//---------------------------------------------------------------------------------------------------------------
//
//  HAUD 2023.03.27
//
//  TR08
//  - XTS_TRANSPORT_LAYER
//
//  fb_Process
//  - grouping of xts stations to sync start process
//  - nFirst to nLast xts stations are checked for starting process simultaneously
//  - basic preparation of station target index in PrepareTarget()
//  - handshake with station control for mover transport through station
//
//---------------------------------------------------------------------------------------------------------------
// This SOFTWARE is provided as an Exemple by THE PROVIDER "as is" and "with all faults." THE PROVIDER makes no 
// representations or warranties of any kind concerning the safety, suitability, lack of viruses, inaccuracies, 
// typographical errors, or other harmful components of this SOFTWARE. There are inherent dangers in the use of 
// any software, and you are solely responsible for determining whether this SOFTWARE is compatible with your 
// equipment and other software installed on your equipment. You are also solely responsible for the protection 
// of your equipment and backup of your data, and THE PROVIDER will not be liable for any damages you may suffer 
// in connection with using, modifying, or distributing this SOFTWARE.
//---------------------------------------------------------------------------------------------------------------
FUNCTION_BLOCK fb_Process IMPLEMENTS I_ExternControl_Process
VAR
  _eType                      : E_PROCESS_TYPE;   // types of process: SINGLE, PARALLEL, SERIAL, DISTRIBUTOR
  _sCheck                     : STRING;

  _eProcessCmd                : E_STATION_CTRL;   // control from property
  _eProcessState              : E_STATION_STATE;  // state   to   property

  {attribute 'displaymode':='bin'}
  _wEnableProcess             : DWORD; // control sets bits to switch on stations
  _bEnabledStation            : POINTER TO ARRAY[1..XTS_Parameter.MAX_STATION]  OF BOOL; // information about all enabled xts stations

  // xts stations
  _stCtrl                     : POINTER TO ARRAY[1..XTS_Parameter.MAX_STATION]  OF ST_STATION_CTRL;
  _stState                    : POINTER TO ARRAY[1..XTS_Parameter.MAX_STATION]  OF ST_STATION_STATE;

  // who is included in process
  // _nFirst to _nLast MUST be in closed consecutive order
  _nStation,
  _nStationCount,
  _nFirstStation,
  _nLastStation               : UINT;

  // work vars for writing onto _stCtrl[nStation].nTargetStation
  _nTarget,
  _nFirstTarget,
  _nLastTarget                : UINT;   // for parallel process xts stations and the last xts station in serial process

  _nSerialTarget              : ARRAY[1..XTS_Parameter.MAX_STATION]  OF UINT; // serial targets within process

  _nPreparedTarget            : ARRAY[1..XTS_Parameter.MAX_MOVER]  OF UINT;   // targets for parallel and single process

  // bitmasks for station states in CycleStation()
  {attribute 'displaymode':='bin'}
  _wEnable                    : DWORD;   // commanded enable of xts station
  {attribute 'displaymode':='bin'}
  _wEnter                     : DWORD;   // mover asking for entry into xts station
  {attribute 'displaymode':='bin'}
  _wStart                     : DWORD;   // xts station asking for process handshake
  {attribute 'displaymode':='bin'}
  _wLeave                     : DWORD;   // xts station wants to send out mover
  {attribute 'displaymode':='bin'}
  _wQueue                     : DWORD;   // mover was entered into xts station list
  {attribute 'displaymode':='bin'}
  _wMoverInStation            : DWORD;   // mover entry was granted, mover is now in station
  {attribute 'displaymode':='bin'}
  _wError                     : DWORD;   // minor error, must be fixed by _stCtrl[nStation]
  {attribute 'displaymode':='bin'}
  _wErrorFatal                : DWORD;   // fatal error, must be fixed by debugging
  {attribute 'displaymode':='bin'}
  _wTargetId                  : DWORD;   // nTargetStation > 0 in _stDtrl[nStation].nTargetStation

  {attribute 'displaymode':='bin'}
  _TargetMask                 : DWORD;   // bit positions correspond to index of xts station
 
  _bNext                      : BOOL;

  _nProcessPerMinute          : uint; // sum of all xts stations output per minute in process
  _rtrigProcess               : ARRAY[1..XTS_Parameter.MAX_STATION] OF Tc2_Standard.R_TRIG;
  _tonPartsPerMinute          : Tc2_Standard.TON;

  _nMoverPerMinute            : POINTER TO ARRAY[1..XTS_Parameter.MAX_STATION]  OF UINT;
  _nMoverCount,
  _nMoverCountOld             : ARRAY[1..XTS_Parameter.MAX_STATION]  OF UINT;

  _eDistributorTarget         : E_PROGRESS;

END_VAR

METHOD private Check : BOOL

IF (_nFirstStation < 1) OR
   (_nFirstStation > MAX_STATION)
THEN
  _sCheck                     := '_nFirstStation out of bounds';
  RETURN;
END_IF

IF (_nLastStation < 1) OR
   (_nLastStation > MAX_STATION)
THEN
  _sCheck                     := '_nLastStation out of bounds';
  RETURN;
END_IF

IF (_nFirstTarget < 1) OR
   (_nFirstTarget > MAX_STATION)
THEN
  _sCheck                     := '_nFirstTarget out of bounds';
  RETURN;
END_IF

IF (_nLastTarget < 1) OR
   (_nLastTarget > MAX_STATION)
THEN
  _sCheck                     := '_nLastTarget out of bounds';
  RETURN;
END_IF

IF NOT (_stCtrl  <> 0)
THEN
  _sCheck                     := '_stCtrl: missing pointer';
  RETURN;
END_IF

IF NOT (_stState <> 0)
THEN
  _sCheck                     := '_stState: missing pointer';
  RETURN;
END_IF

IF NOT (_bEnabledStation  <> 0)
THEN
  _sCheck                     := '_bEnableStation: missing pointer';
  RETURN;
END_IF

IF not (_nMoverPerMinute <> 0)
THEN
  _sCheck                     := '_nMoverPerMinute: missing pointer';
  RETURN;
END_IF

_nStationCount                := _nLastStation - _nFirstStation + 1;

IF (_nStationCount < 1) OR
   (_nStationCount > (SIZEOF(WORD)*8))
THEN
  _sCheck                     := '_nStationCount out of bounds';
  RETURN;
END_IF


_sCheck                       := TO_STRING(E_PROGRESS.PROGRESS_DONE);
Check                         := TRUE;
END_METHOD

METHOD Cycle
VAR_INST
  _nStn     : uint;
END_VAR
IF NOT Check() THEN RETURN; END_IF


//-----------------------------------------------------------------------------
// collect state information from xts stations
// state information is collected in Masks (WORD), 
// every bit represents one XTS station in process
//-----------------------------------------------------------------------------
//  _wEnable                        : enable cmd was given to xts station
//  _wEnter                         : a mover is requesting entry
//  _wStart                         : mover has arrived and xts station is ready
//  _wLeave                         : xts station wants to send mover out
//  _wQueue                         : somebody's waiting
//  _wMoverInStation                : mover is in station
//  _wError                         : error state for handshake
//  _wErrorFatal                    : error state for severe problems (debugging required)
//  _wTargetId                      : Ctrl.nTargetStation > 0
//  _wMoverInQueueSerial            : SERIAL process: bits to check whether a mover is waiting to be processed
//
CycleStation();                     // get state information from all XtsStations in process
//-----------------------------------------------------------------------------
//-----------------------------------------------------------------------------
//  E_STATION_CTRL.STATION_INIT: hard reset of process and XtsStations
//-----------------------------------------------------------------------------
CASE _eProcessCmd                   // check input property
OF
  E_STATION_CTRL.STATION_INIT:      // commanded init from ctrl
    CASE _eType
    OF
      E_PROCESS_TYPE.SERIAL:
        InitSerialTargets();
    END_CASE
    Init();                         RETURN; // rest you will, return you must
END_CASE
//-----------------------------------------------------------------------------
// E_STATION_STATE.STATION_INIT: pass through here and switch off XtsStations
//-----------------------------------------------------------------------------
CASE _eProcessState                 // check output property
OF
  E_STATION_STATE.STATION_INIT:     // xts station empty, disabled by default
    _eProcessState                  := E_STATION_STATE.STATION_DISABLE;
    FOR _nStn := _nLastStation TO _nFirstStation BY(-1) 
    DO
      _stCtrl^[_nStn].eCmd          := E_STATION_CTRL.STATION_DISABLE;
    END_FOR

END_CASE
//-----------------------------------------------------------------------------
//  E_STATION_STATE.STATION_DISABLE: wait for enable from flow control
//-----------------------------------------------------------------------------
CASE _eProcessState                 // check output property
OF
  E_STATION_STATE.STATION_DISABLE:  // check for enable command
    IF (_eProcessCmd = E_STATION_CTRL.STATION_ENABLE)
    THEN
      _eProcessState                := E_STATION_STATE.STATION_ENABLE;

      FOR _nStn := _nLastStation TO _nFirstStation BY(-1) 
      DO
          _stCtrl^[_nStn].eCmd      := E_STATION_CTRL.STATION_ENABLE;
      END_FOR
    END_IF
END_CASE
//-----------------------------------------------------------------------------
//  E_STATION_STATE.STATION_ENABLE: check Cmd and wait for XtsStations to be enabled
//-----------------------------------------------------------------------------
CASE _eProcessState
OF
  E_STATION_STATE.STATION_ENABLE:
    CASE _eProcessCmd
    OF
      E_STATION_CTRL.STATION_DISABLE:
        _eProcessState              := E_STATION_STATE.STATION_INIT;

      E_STATION_CTRL.STATION_ENABLE:
        IF (_wEnable = _wEnableProcess)
        THEN
          InitSerialTargets();
          _eProcessState            := E_STATION_STATE.STATION_DETECT_MOVER;
        END_IF
    END_CASE
END_CASE
//-----------------------------------------------------------------------------
// E_STATION_STATE.STATION_DETECT_MOVER: wait for any XtsStation to 
//                                       have a mover ready to enter
//-----------------------------------------------------------------------------
CASE _eProcessState
OF
  E_STATION_STATE.STATION_DETECT_MOVER:
    CASE _eProcessCmd
    OF
      E_STATION_CTRL.STATION_DISABLE:
        _eProcessState              := E_STATION_STATE.STATION_INIT;

      E_STATION_CTRL.STATION_ENABLE:
        IF (_wEnter > 0)            // at least one mover is asking for entry
        THEN
          _eDistributorTarget       := E_PROGRESS.PROGRESS_INVALID;

                                    // switch process state in order to tell process control
          _eProcessState            := E_STATION_STATE.STATION_MOVER_ENTER;
        END_IF
    END_CASE
END_CASE
//-----------------------------------------------------------------------------
//  E_STATION_STATE.STATION_MOVER_ENTER: check if infeed conditions are met, 
//                                       depending on type of process
//                                       Cmd from input (flow control)
//-----------------------------------------------------------------------------
CASE _eProcessState
OF
  E_STATION_STATE.STATION_MOVER_ENTER:
    CASE _eProcessCmd               // check input property
    OF
      E_STATION_CTRL.STATION_DISABLE:
        _eProcessState              := E_STATION_STATE.STATION_INIT;

      E_STATION_CTRL.STATION_MOVER_ENTER:
        FOR _nStn := _nLastStation TO _nFirstStation BY(-1) 
        DO
          CASE _stState^[_nStn].eState
          OF
          E_STATION_STATE.STATION_MOVER_ENTER,
          E_STATION_STATE.STATION_MOVER_IN_TARGET,
          E_STATION_STATE.STATION_PROCESS_START:
            IF GetBitDWord(_wEnter, (_nStn - _nFirstStation))
            THEN
              _stCtrl^[_nStn].eCmd  := E_STATION_CTRL.STATION_MOVER_ENTER;
            END_IF
          END_CASE
        END_FOR

        CASE _eType
        OF
          E_PROCESS_TYPE.PARALLEL_STRICT:
            IF (_wStart = _wEnable) // all who are enabled must have mover, in order to continue
            THEN
              _eProcessState        := E_STATION_STATE.STATION_PROCESS_START;
            END_IF

          E_PROCESS_TYPE.PARALLEL: 
            IF (_wStart = _wEnter)
            THEN
              _eProcessState        := E_STATION_STATE.STATION_PROCESS_START;
            END_IF

          E_PROCESS_TYPE.SERIAL:    // all who have work to do must have mover, in order to continue
            IF (_wMoverInStation > 0)
            THEN
              IF (_wStart = _wMoverInStation)
              THEN
                _eProcessState      := E_STATION_STATE.STATION_PROCESS_START;
              END_IF
            END_IF
        ELSE
          _eProcessState            := E_STATION_STATE.STATION_PROCESS_START;
        END_CASE

      E_STATION_CTRL.STATION_MOVER_SEND:  // flow control decided to skip process
        FOR _nStn := _nLastStation TO _nFirstStation BY(-1) 
        DO
          IF _bEnabledStation^[_nStn] AND 
             GetBitDWord(_wQueue, (_nStn-_nFirstStation))
          THEN
            IF (_TargetMask > 0)
            THEN
              // station is enabled AND has a mover in Queue to send
              _stCtrl^[_nStn].eCmd    := E_STATION_CTRL.STATION_MOVER_SEND;
            END_IF
          END_IF
        END_FOR
        IF (_wLeave > 0)            // wait for XtsStation to switch to outfeed
        THEN
          IF (_TargetMask > 0)
          THEN
            _eDistributorTarget       := DistributorTarget(_TargetMask);         // prepare target for mover
            IF (_eDistributorTarget = E_PROGRESS.PROGRESS_DONE)
            THEN
              _wStart                 := _wLeave;
              _eProcessState          := E_STATION_STATE.STATION_CHECK;
            END_IF
          END_IF
        END_IF 
    END_CASE
END_CASE
//-----------------------------------------------------------------------------
// synced process handshake on all stations in process
//-----------------------------------------------------------------------------
CASE _eProcessState                 // check output property
OF
  E_STATION_STATE.STATION_PROCESS_START:
    CASE _eType                     // decision for synced start varies for e_process_type
    OF
      E_PROCESS_TYPE.SERIAL:        // serial process must have had a mover waiting, which is now processed
      CASE _eProcessCmd             // check command input property
      OF
        E_STATION_CTRL.STATION_PROCESS_START,
        E_STATION_CTRL.STATION_PROCESS_DONE:
            IF (_wStart = _wMoverInStation)
            THEN
              _eProcessState          := E_STATION_STATE.STATION_PROCESS_DONE;
              FOR _nStn := _nLastStation TO _nFirstStation BY(-1) 
              DO
                // check for correct state on XtsStation
                CASE _stState^[_nStn].eState
                OF
                E_STATION_STATE.STATION_PROCESS_START:
                  _stCtrl^[_nStn].eCmd  := _eProcessCmd;
                END_CASE
              END_FOR
            END_IF
      END_CASE
    ELSE
      CASE _eProcessCmd             // check command input property
      OF
        E_STATION_CTRL.STATION_PROCESS_START,
        E_STATION_CTRL.STATION_PROCESS_DONE:
          IF (_wStart = _wEnter)
          THEN
            _eProcessState          := E_STATION_STATE.STATION_PROCESS_DONE;
            FOR _nStn := _nLastStation TO _nFirstStation BY(-1) 
            DO
              // check for correct state on XtsStation
              CASE _stState^[_nStn].eState
              OF
              E_STATION_STATE.STATION_PROCESS_START:
                _stCtrl^[_nStn].eCmd  := _eProcessCmd;
              END_CASE
            END_FOR
          END_IF
      END_CASE
    END_CASE
END_CASE
//-----------------------------------------------------------------------------
// synced process handshake on all stations in process
//-----------------------------------------------------------------------------
CASE _eProcessState                 // check output property
OF
  E_STATION_STATE.STATION_PROCESS_DONE:
    CASE _eProcessCmd               // check command input property
    OF
      E_STATION_CTRL.STATION_PROCESS_DONE: 
        FOR _nStn := _nLastStation TO _nFirstStation BY(-1) 
        DO
          _stCtrl^[_nStn].eCmd      := E_STATION_CTRL.STATION_PROCESS_DONE;
        END_FOR
        IF (_wLeave > 0)            // _wLeave tells us that xts station has mover to send
        THEN
          CASE _eType
          OF
            E_PROCESS_TYPE.SERIAL:
              _eProcessState        := E_STATION_STATE.STATION_CHECK;
              IF (_stState^[_nLastStation].nMoverId > 0)
              THEN
                PrepareLastSerialTarget();     // target for last xts station in serial process
              END_IF
    
              FOR _nStn := (_nLastStation - 1) TO _nFirstStation BY(-1) 
              DO
                _stCtrl^[_nStn].nTargetStation    := TO_USINT(_nSerialTarget[_nStn]);
              END_FOR
          ELSE
              IF (_TargetMask > 0)
              THEN
                ParallelTargets(_TargetMask);
                _eProcessState      := E_STATION_STATE.STATION_CHECK;
              END_IF
          END_CASE
        END_IF
    END_CASE
END_CASE
//-----------------------------------------------------------------------------
//-----------------------------------------------------------------------------
CASE _eProcessState
OF
  E_STATION_STATE.STATION_CHECK:    // TODO: implement procedure for target plausibility
    IF (_wTargetId > 0)             // simple check any target before switching to outfeed
    THEN
       _eProcessState               := E_STATION_STATE.STATION_MOVER_OUT;
(*
    ELSE                            // in case of invalid target, wait here for retry
      CASE _eType                   // retry varies for e_process_type
      OF
        E_PROCESS_TYPE.DISTRIBUTOR:
          IF (_eProcessCmd = E_STATION_CTRL.STATION_ENABLE)
          THEN
            // only distributor can land here directly; retry mover infeed
            _eProcessState          := E_STATION_STATE.STATION_MOVER_ENTER;
          END_IF
      ELSE
          IF (_eProcessCmd = E_STATION_CTRL.STATION_PROCESS_START)
          THEN
            // all other e_process_type must go back to process handshake
            _eProcessState          := E_STATION_STATE.STATION_PROCESS_DONE;
          END_IF
      END_CASE
*)
    END_IF
END_CASE
//-----------------------------------------------------------------------------
//-----------------------------------------------------------------------------
CASE _eProcessState
OF
  E_STATION_STATE.STATION_MOVER_OUT:
    IF (_wLeave = 0)                // all movers are gone
    THEN
      _eProcessState                := E_STATION_STATE.STATION_MOVER_GONE;

    ELSIF (_wLeave = _wStart)       // wait for everybody to be ready for send out
    THEN
      IF (_eProcessCmd = E_STATION_CTRL.STATION_MOVER_OUT)
      THEN
        FOR _nStn := _nLastStation TO _nFirstStation BY(-1) 
        DO
          CASE _stState^[_nStn].eState  // double check valid xts station state
          OF
            E_STATION_STATE.STATION_MOVER_OUT:
              IF (_stCtrl^[_nStn].nTargetStation > 0) // double check ticket on ctrl struct
              THEN
                _stCtrl^[_nStn].eCmd  := E_STATION_CTRL.STATION_MOVER_OUT;
              END_IF
          END_CASE
        END_FOR
      END_IF
    END_IF
END_CASE
//-----------------------------------------------------------------------------
//-----------------------------------------------------------------------------
CASE _eProcessState
OF
  E_STATION_STATE.STATION_MOVER_GONE:   // station is empty, quit mover gone and go back to the beginning
    FOR _nStn := _nLastStation TO _nFirstStation BY(-1) 
    DO
      _stCtrl^[_nStn].nTargetStation := 0;
      _stCtrl^[_nStn].eCmd      := E_STATION_CTRL.STATION_MOVER_GONE;
    END_FOR
    _eProcessState              := E_STATION_STATE.STATION_INIT;
END_CASE
END_METHOD

METHOD PRIVATE CycleStation
VAR
  _k                  : UINT;
END_VAR
IF NOT Check() THEN RETURN; END_IF

_wError                                   :=
_wErrorFatal                              := 0;

FOR _nStation := _nLastStation TO _nFirstStation BY(-1) 
DO
  // copy bit for enable station from input word to global array in GVL_PROCESS,
  //  - other processes read enabled state on mover out (PrepareTarget)
  _bEnabledStation^[_nStation]            := GetBitDWord(_wEnableProcess, (_nStation-_nFirstStation));

  IF (_stCtrl^[_nStation].nTargetStation > 0)
  THEN
    _wTargetId                            := SetBitDWord(_wTargetId,  (_nStation-_nFirstStation));
  ELSE
    _wTargetId                            := DelBitDWord(_wTargetId,  (_nStation-_nFirstStation));
  END_IF

  IF (_stState^[_nStation].nMoverId > 0)
  THEN
    _wMoverInStation                      := SetBitDWord(_wMoverInStation,  (_nStation-_nFirstStation));
  ELSE
    _wMoverInStation                      := DelBitDWord(_wMoverInStation,  (_nStation-_nFirstStation));
  END_IF

  IF (_stState^[_nStation].nQueue > 0)
  THEN
    _wQueue                               := SetBitDWord(_wQueue,  (_nStation-_nFirstStation));
  ELSE
    _wQueue                               := DelBitDWord(_wQueue,  (_nStation-_nFirstStation));
  END_IF

  CASE _stCtrl^[_nStation].eCmd
  OF
    E_STATION_CTRL.STATION_INIT:
      _stCtrl^[_nStation].nTargetStation  := 0;
      _wEnable                            := DelBitDWord(_wEnable, (_nStation-_nFirstStation));
      _wEnter                             := DelBitDWord(_wEnter,  (_nStation-_nFirstStation));
      _wStart                             := DelBitDWord(_wStart,  (_nStation-_nFirstStation));
      _wLeave                             := DelBitDWord(_wLeave,  (_nStation-_nFirstStation));

    E_STATION_CTRL.STATION_ENABLE:
      _wEnable                            := SetBitDWord(_wEnable, (_nStation-_nFirstStation));
  END_CASE

  CASE _stState^[_nStation].eState
  OF
    E_STATION_STATE.STATION_DISABLE:
      _wEnter                             := DelBitDWord(_wEnter,  (_nStation-_nFirstStation));

    E_STATION_STATE.STATION_MOVER_ENTER,
    E_STATION_STATE.STATION_MOVER_IN_TARGET:
      _wEnter                             := SetBitDWord(_wEnter,  (_nStation-_nFirstStation));
  
    E_STATION_STATE.STATION_PROCESS_START,
    E_STATION_STATE.STATION_PROCESS_DONE:
      _wStart                             := SetBitDWord(_wStart,  (_nStation-_nFirstStation));
  
    E_STATION_STATE.STATION_MOVER_OUT:
      _wLeave                             := SetBitDWord(_wLeave,  (_nStation-_nFirstStation));


    E_STATION_STATE.STATION_MOVER_GONE:
      _stCtrl^[_nStation].nTargetStation  := 0;
      _wStart                             := DelBitDWord(_wStart,  (_nStation-_nFirstStation));
      _wLeave                             := DelBitDWord(_wLeave,  (_nStation-_nFirstStation));
      _wEnable                            := DelBitDWord(_wEnable, (_nStation-_nFirstStation));
      _wEnter                             := DelBitDWord(_wEnter,  (_nStation-_nFirstStation));


    E_STATION_STATE.STATION_ERROR_LIST_STATION_ID_WRONG,  // wrong station ID in mover ticket (nTargetId written by preceeding station/process)
    E_STATION_STATE.STATION_ERROR_OUTFEED_TARGET_INVALID, // write correct target on station Ctrl.nTargetStation
    E_STATION_STATE.STATION_ERROR_INFEED_ERROR,           // clear mover error via Ctrl/State interface and retry on XTS station directly
    E_STATION_STATE.STATION_ERROR_OUTFEED_ERROR:          // clear mover error via Ctrl/State interface and retry on XTS station directly
      _wError                             := SetBitDWord(_wError,      (_nStation-_nFirstStation));

    E_STATION_STATE.STATION_ERROR_FATAL:
      _wErrorFatal                        := SetBitDWord(_wErrorFatal, (_nStation-_nFirstStation));

  END_CASE
END_FOR


_nProcessPerMinute          := 0;
// get mover counter
FOR _k := _nLastStation TO _nFirstStation BY(-1) 
DO
  _rtrigProcess[_k](
                  CLK       := (_stCtrl^[_k].eCmd = E_STATION_CTRL.STATION_MOVER_OUT));

  IF _rtrigProcess[_k].Q
  THEN
    _nMoverCount[_k]        := _nMoverCount[_k] + 1;
  END_IF
  
  IF _tonPartsperMinute.Q
  THEN
    _nMoverPerMinute^[_k]   := _nMoverCount[_k] - _nMoverCountOld[_k];
    _nMoverCountOld  [_k]   := _nMoverCount[_k];
  END_IF
  _nProcessPerMinute        := _nProcessPerMinute + _nMoverPerMinute^[_k]; 
END_FOR

IF _tonPartsperMinute.q
THEN
  _tonPartsperMinute(
                  IN        :=FALSE);
END_IF

_tonPartsperMinute(
                  IN        := TRUE, 
                  PT        := T#60S);
END_METHOD

METHOD PUBLIC DelBitDWord : DWORD
VAR_INPUT
  inVal   : DWORD;
  bitNo   : DWORD;
END_VAR
VAR
  wConst : DWORD := 1;
END_VAR
IF ( inVal AND SHL( wConst,bitNo MOD 16 ) ) > 0 THEN
  DelBitDWord := inVal XOR (SHL( wConst,bitNo MOD 16 ));
ELSE
  DelBitDWord := inVal;
END_IF
END_METHOD

METHOD DistributorTarget : e_progress
VAR_INPUT
  wTarget         : DWORD; // bits for target stations to be used
END_VAR
VAR_INST
  _eResult        : E_PROGRESS;
  {attribute 'displaymode':='bin'}
  _wtg            : DWORD;
END_VAR
IF NOT Check() THEN RETURN; END_IF
_wtg := wTarget;

// check if target station is enabled
IF GetBitDWord(wTarget, (_nTarget))
THEN
  _nPreparedTarget[_stState^[_nFirstStation].nMoverId]  := _nLastTarget - _nTarget;
  _stCtrl^[_nFirstStation].nTargetStation               := TO_USINT(_nLastTarget - _nTarget);
  _eResult                                              := E_PROGRESS.PROGRESS_DONE;
ELSE
  _eResult                                              := e_progress.PROGRESS_BUSY;
END_IF

_nTarget                      := _nTarget + 1;
IF (_nLastTarget - _nTarget < _nFirstTarget)
THEN
  _nTarget                    := 0;
END_IF

DistributorTarget                                       := _eResult;
END_METHOD

PROPERTY EnabledStation : POINTER TO ARRAY[1..XTS_Parameter.MAX_STATION]  OF bool;
SET
_bEnabledStation := EnabledStation;
END_SET
END_PROPERTY

PROPERTY EnableProcess : dword
GET
EnableProcess := _wEnableProcess;
END_GET
SET
_wEnableProcess := EnableProcess;
END_SET
END_PROPERTY

METHOD PUBLIC GetBitDWord : BOOL
VAR_INPUT
  inVal   : DWORD;
  bitNo   : DINT;
END_VAR
VAR
  wConst : DWORD := 1;
END_VAR
IF ( inVal AND SHL( wConst,DINT_TO_SINT(bitNo) MOD 32 ) ) > 0
THEN
  GetBitDWord := TRUE;
ELSE
  GetBitDWord := FALSE;
END_IF
END_METHOD

METHOD PUBLIC Init : BOOL
VAR
  _nStn     : UINT;
END_VAR
IF NOT (_nLastStation   > 0) OR
   NOT (_nFirstStation  > 0) OR
   NOT (_nLastStation   < MAX_STATION+1) OR
   NOT (_nFirstStation  < MAX_STATION+1)
THEN
  Init := FALSE;
  _eProcessState                := E_STATION_STATE.STATION_NO_INIT;
ELSE
  _eProcessState                := E_STATION_STATE.STATION_NO_INIT;

  FOR _nStn := _nLastStation TO _nFirstStation BY(-1) 
  DO
    _stCtrl^[_nStn].eCmd        := E_STATION_CTRL.STATION_INIT;
    _stCtrl^[_nStn].nMask       := 0;

    IF NOT (_stState^[_nStn].eState = E_STATION_STATE.STATION_INIT)
    THEN
      Init := FALSE;
      RETURN;
    END_IF  
  END_FOR

  memset(ADR(_nMoverCount),       0, SIZEOF(_nMoverCount));
  memset(ADR(_nMoverCountOld),    0, SIZEOF(_nMoverCountOld));
  _nTarget                      := 0;

  _eProcessState                := E_STATION_STATE.STATION_INIT;

  Init := TRUE;
END_IF
END_METHOD

METHOD PRIVATE InitSerialTargets
VAR
  _k    : uint;
END_VAR

IF NOT (_nStationCount > 1)
THEN
  RETURN;
END_IF

// serial process must always have at least two xts stations to work with
FOR _nStation := _nLastStation TO _nFirstStation+1 BY(-1) 
DO
  IF (_bEnabledStation^[_nStation])
  THEN
    _nSerialTarget[_nStation-1] := _nStation;
  END_IF
END_FOR
END_METHOD

PROPERTY MoverCountInQueue : uint
GET
VAR
  _nTmp   : UINT;
  _nCount : uint;
END_VAR
IF NOT (_nStationCount > 0)
THEN
  MoverCountInQueue := 0;
  RETURN;
END_IF

FOR _nTmp := _nLastStation TO _nFirstStation BY(-1)
DO
  _nCount := _nCount + _stState^[_nTmp].nQueue;
END_FOR

MoverCountInQueue := _nCount;
END_GET
END_PROPERTY

PROPERTY MoverInQueue : Bool
GET
MoverInQueue  := SEL((_wQueue > 0), FALSE, TRUE);
END_GET
END_PROPERTY

PROPERTY MoverPerMinute : pointer to ARRAY[1..XTS_Parameter.MAX_STATION]  OF UINT
SET
_nMoverPerMinute  := MoverPerMinute;
END_SET
END_PROPERTY

METHOD PRIVATE ParallelTargets : E_PROGRESS
VAR_INPUT
  wTarget         : DWORD; // bits for target stations to be used
END_VAR
VAR_INST
  {attribute 'displaymode':='bin'}
  _wtg            : DWORD;
  _nt,
  _idxStation     : UINT;
END_VAR
IF NOT Check() THEN RETURN; END_IF
_wtg := wTarget;


FOR _idxStation := _nLastStation TO _nFirstStation BY(-1) 
DO
  _nt                           := _nLastTarget - _nTarget;

  // check if target station is enabled
  IF GetBitDWord(wTarget, (_nTarget))
  THEN
    IF (_stState^[_idxStation].nMoverId <> 0)
    THEN
      _nPreparedTarget[_stState^[_idxStation].nMoverId]  := _nt;
      _stCtrl^[_idxStation].nTargetStation               := TO_USINT(_nt);
    END_IF
  END_IF

  _nTarget                      := _nTarget + 1;
  IF (_nLastTarget - _nTarget < _nFirstTarget)
  THEN
    _nTarget                    := 0;
  END_IF
END_FOR
END_METHOD

METHOD PRIVATE PrepareLastSerialTarget
VAR
  _nt   : uint;
END_VAR

_nt                           := _nLastTarget - _nTarget;
_nTarget                      := _nTarget + 1;

// check if target station is enabled
IF (_bEnabledStation^[_nt])
THEN
  _nPreparedTarget[_stState^[_nLastStation].nMoverId]  := _nt;
  _stCtrl^[_nLastStation].nTargetStation               := TO_USINT(_nt);
END_IF

IF (_nLastTarget - _nTarget < _nFirstTarget)
THEN
  _nTarget                    := 0;
END_IF
END_METHOD

PROPERTY ProcessCmd : E_STATION_CTRL
SET
_eProcessCmd := ProcessCmd;
END_SET
END_PROPERTY

PROPERTY ProcessPerMinute : uint
GET
ProcessPerMinute := _nProcessPerMinute;
END_GET
END_PROPERTY

PROPERTY ProcessState : E_STATION_STATE
GET
ProcessState := _eProcessState;
END_GET
END_PROPERTY

PROPERTY ProcessType : e_process_type
GET
ProcessType := _eType;
END_GET
SET
_eType := ProcessType;
END_SET
END_PROPERTY

METHOD PUBLIC SetBitDWord : DWORD
VAR_INPUT
  inVal   : DWORD;
  bitNo   : DWORD;
END_VAR
VAR
  wConst  : DWORD := 1;
END_VAR
SetBitDWord := inVal OR SHL( wConst,bitNo MOD 32 );
END_METHOD

METHOD PUBLIC SetBitWord : WORD
VAR_INPUT
  inVal   : WORD;
  bitNo   : DINT;
END_VAR
VAR
  wConst  : WORD := 1;
END_VAR
SetBitWord := inVal OR SHL( wConst,bitNo MOD 16 );
END_METHOD

PROPERTY StationCount : uint
GET
StationCount := _nStationCount;
END_GET
END_PROPERTY

PROPERTY StationCtrl : pointer to ARRAY[1..XTS_Parameter.MAX_STATION]  OF ST_STATION_CTRL;
SET
_stCtrl := StationCtrl;
END_SET
END_PROPERTY

PROPERTY StationFirst : uint
GET
StationFirst := _nFirstStation;
END_GET
SET
_nFirstStation := StationFirst;
END_SET
END_PROPERTY

PROPERTY StationLast : uint
GET
StationLast := _nLastStation;
END_GET
SET
_nLastStation := StationLast;
END_SET
END_PROPERTY

PROPERTY StationState : POINTER TO ARRAY[1..XTS_Parameter.MAX_STATION]  OF ST_STATION_STATE
SET
_stState := StationState;
END_SET
END_PROPERTY

PROPERTY TargetFirst : uint
GET
TargetFirst := _nFirstTarget;
END_GET
SET
_nFirstTarget := TargetFirst;
END_SET
END_PROPERTY

PROPERTY TargetLast : uint
GET
TargetLast := _nLastTarget;
END_GET
SET
_nLastTarget := TargetLast;
END_SET
END_PROPERTY

PROPERTY TargetMask : dword
GET
TargetMask := _TargetMask;
END_GET
SET
_TargetMask := TargetMask;
END_SET
END_PROPERTY

END_FUNCTION_BLOCK

(* stored: Version 1.1.0.1, ProductVersion 3.1.4024.12
   POU fb_Process: Id {da86ec44-e899-45cb-8522-c0f7a497324a}, SpecialFunc None
   Folder private: Id {ef591d19-6a22-400f-80f2-48bce4f2b2eb}
   Folder properties: Id {00319e58-6c2c-4aca-bec4-fee440d08884}
   Folder public: Id {7e97a5cb-3ed9-40d2-992f-cb7c96292b31}
   Method Check: Id {229e5281-97c6-4cad-b72d-bce792434909}
   Method Cycle: Id {5d9343b9-7566-4654-850b-142338388e5d}
   Method CycleStation: Id {009c99bc-3f0f-48cb-9438-eb4d90e6d4d0}
   Method DelBitDWord: Id {2fd93023-4323-4a27-9876-b223c0f7241e}
   Method DistributorTarget: Id {10dcb0c8-4c69-4b0e-9499-245d0f9de438}
   Property EnabledStation: Id {fab1679f-d362-4221-adb9-88cee6e9e6d7}
   Set Set: Id {059cc7ea-6bda-4b61-b086-a7ba6cdc895a}
   Property EnableProcess: Id {7c790d0b-a53d-40bf-b6bd-1c4cc587158d}
   Get Get: Id {0874ed85-5165-412e-903a-1e28fd1e2715}
   Set Set: Id {05a75b91-4880-4efd-a0da-62e3a72730d1}
   Method GetBitDWord: Id {c24075ee-d4b4-4f17-b387-ca667f5b9cbb}
   Method Init: Id {cb35fdde-b84e-42f2-be27-a7e2dfc72e31}
   Method InitSerialTargets: Id {64fc78a5-5a07-420a-b6a4-803be9ca4d52}
   Property MoverCountInQueue: Id {1f60161d-c3f4-421c-af40-3538902ebcbd}
   Get Get: Id {26f04c33-31b3-4607-8368-38a23734ca22}
   Property MoverInQueue: Id {4541e140-57cd-430b-8fae-fbf6cf35ed52}
   Get Get: Id {ae78173a-6d76-4d3e-958f-44ac060b4b9b}
   Property MoverPerMinute: Id {a5633af1-33d3-43c1-a7f0-451b802e11f3}
   Set Set: Id {8d4f204a-a28d-4021-8cea-647c6ad83f5d}
   Method ParallelTargets: Id {1b573a2b-9344-4048-b386-4f42ea4f4f85}
   Method PrepareLastSerialTarget: Id {3cfabe49-4c49-457f-bc75-f3d8da2c1c43}
   Property ProcessCmd: Id {ec10d53d-6811-4d32-84d4-4b2023aac397}
   Set Set: Id {3d1daf29-0ad9-44fa-a352-15dc67b0c2a1}
   Property ProcessPerMinute: Id {816e0b83-e712-4dd6-8776-81f0599e0165}
   Get Get: Id {2d7dadfb-d25e-47b9-a733-edd3cab3ea45}
   Property ProcessState: Id {391db9ce-ac85-4c5f-8c47-7d975024be6c}
   Get Get: Id {5a79982c-bb54-48ed-b038-237d4cfe1f32}
   Property ProcessType: Id {8a7517ef-08e9-4495-84fb-4434c68a463b}
   Get Get: Id {b4aacb1c-401a-431f-a3ff-93a14ed467de}
   Set Set: Id {9625e2c1-c262-476e-a53c-7bf800aaa2f3}
   Method SetBitDWord: Id {07820c7b-9331-49b5-89a4-719feb5594f7}
   Method SetBitWord: Id {a2527f69-a904-46eb-87b3-a348014b22dc}
   Property StationCount: Id {3fa6e598-9d0f-4039-9281-d5cfbfd3d26a}
   Get Get: Id {d3917fa2-ae66-47da-a982-c68a259d9cef}
   Property StationCtrl: Id {54f02afe-19e2-4e58-80bb-7dd3c88c31a3}
   Set Set: Id {5b956450-26e7-406c-b2e3-712eb2c09a6b}
   Property StationFirst: Id {14e12906-fcf3-43f0-9320-604e1c488997}
   Get Get: Id {b2c8fd95-49aa-4f95-b623-1e786aa8296d}
   Set Set: Id {23c8506f-8c5d-48d3-b7a8-85e178c0b436}
   Property StationLast: Id {66b1c133-8ea7-425f-a05d-435ec8a6fe75}
   Get Get: Id {78bbb339-c485-4284-8cfa-a1468f5cbbc0}
   Set Set: Id {e0256e78-ee9d-48d9-9468-746a7009e98b}
   Property StationState: Id {12d671ce-4f48-4f2d-801b-f179fe1b4407}
   Set Set: Id {b9409299-2a76-4f7e-ad65-a952bdd1334f}
   Property TargetFirst: Id {f7dee83a-8746-44d0-8747-363a91698d07}
   Get Get: Id {65db5591-8c5e-42b7-afbb-3c1dc0f4e381}
   Set Set: Id {7e76c355-577a-48ba-8b6b-2808053fc746}
   Property TargetLast: Id {da86159d-6ee5-4404-81d4-db749bbb3513}
   Get Get: Id {229070bc-f9cf-4a0c-90aa-62f3bd5d36df}
   Set Set: Id {5bd9be9c-7374-4097-86e8-97f8e4696dc9}
   Property TargetMask: Id {299fb60d-893e-406c-a169-4e5ca2cdd902}
   Get Get: Id {d8bfd69f-a07e-4bb0-a945-c2a3950800c8}
   Set Set: Id {2492d0b1-d603-4be1-85fb-56561e253167} *)
